(* Schneider Machine Expert - Basic project control, file version 2.7.0.0 *)
(* ProjectInformations: Name=Nuevo proyecto *)

HARDWARE
  Cpu 0: TM221M16R/G
  EthernetConfiguration: NetworkName=M221, IpAllocationMode=FixedAddress, IpAddress=0.0.0.0, SubnetMask=0.0.0.0
  SerialLineConfiguration: Baud=Baud19200, Parity=ParityEven, DataBits=DataBits8, StopBits=StopBits1, PhysicalMedium=PhysicalMediumRs485, TransmissionMode=TransmissionModeModbusRtu, SlaveId=1, Addressing=SlaveAddressing
  MastTask: UsePeriodScanMode=true, PeriodScan=10
  FastTask: Period=255
  CpuBehavior: StartingMode=StartAsPreviousState, AutoSaveRamOnEeprom=true, WatchdogPeriod=250

SYMBOLS  (address, symbol, comment, settings)
  %MW0      ER
  %MW10     PRO
  %MW20     INT
  %MW30     ER_ACUM
  %MW40     DER_ERR
  %MW50     DER
  %MW60     ERR_PREV
  %MW100    U_OUT
  %KW1      KP  [Value=4]
  %KW2      KI  [Value=3]
  %KW3      KD  [Value=1]

POU Nuevo POU
  (* SectionNumber=1 *)

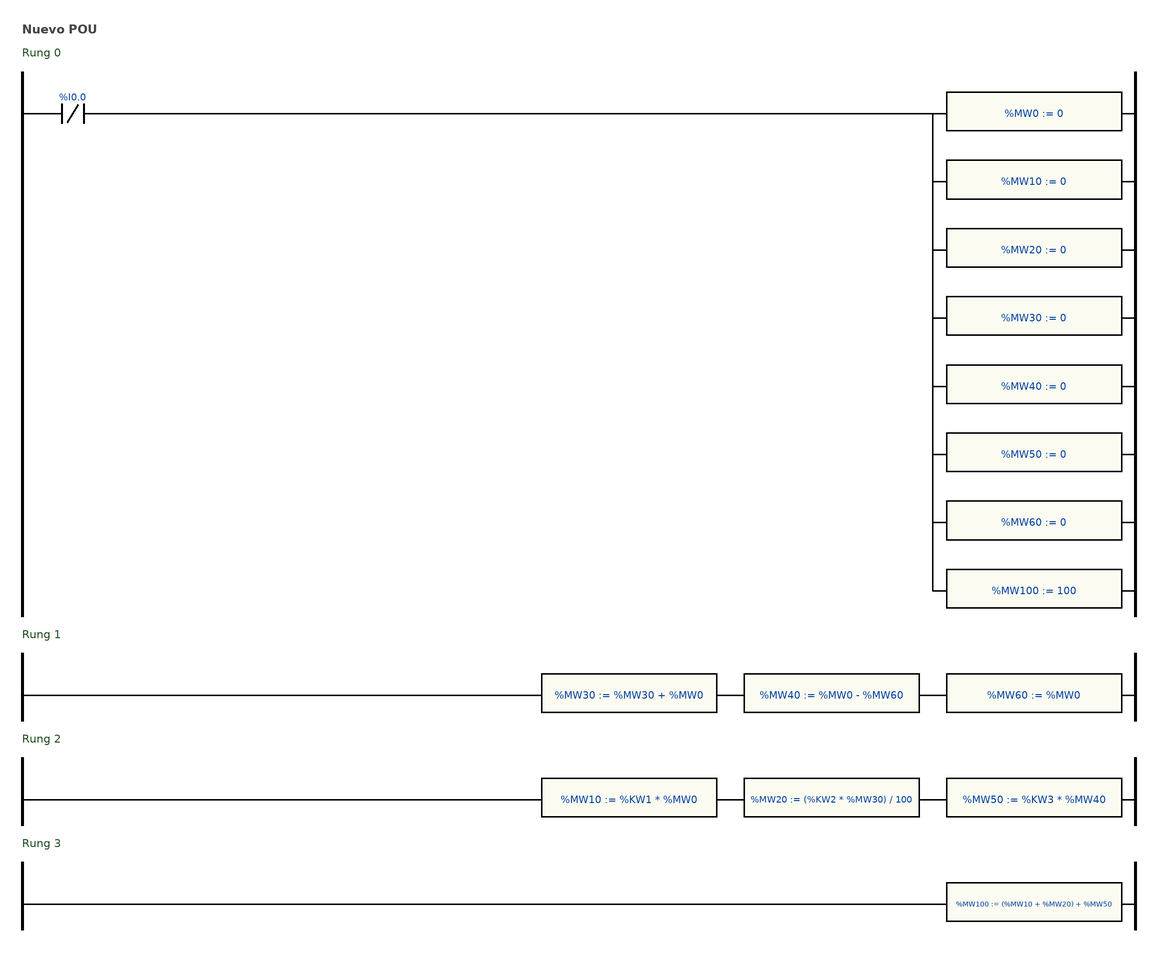

// Rung 0
  LDN %I0.0
  [ %MW0 := 0 ]           (* ER *)
  [ %MW10 := 0 ]          (* PRO *)
  [ %MW20 := 0 ]          (* INT *)
  [ %MW30 := 0 ]          (* ER_ACUM *)
  [ %MW40 := 0 ]          (* DER_ERR *)
  [ %MW50 := 0 ]          (* DER *)
  [ %MW60 := 0 ]          (* ERR_PREV *)
  [ %MW100 := 100 ]       (* U_OUT *)
  // as ST:
  //   IF NOT %I0.0 THEN ER := 0; END_IF;
  //   IF NOT %I0.0 THEN PRO := 0; END_IF;
  //   IF NOT %I0.0 THEN INT := 0; END_IF;
  //   IF NOT %I0.0 THEN ER_ACUM := 0; END_IF;
  //   IF NOT %I0.0 THEN DER_ERR := 0; END_IF;
  //   IF NOT %I0.0 THEN DER := 0; END_IF;
  //   IF NOT %I0.0 THEN ERR_PREV := 0; END_IF;
  //   IF NOT %I0.0 THEN U_OUT := 100; END_IF;

// Rung 1
  LD 1
  OPER [ %MW30 := %MW30 + %MW0 ](* ER_ACUM, ER_ACUM, ER *)
  OPER [ %MW40 := %MW0 - %MW60 ](* DER_ERR, ER, ERR_PREV *)
  [ %MW60 := %MW0 ]       (* ERR_PREV, ER *)
  // as ST:
  //   ER_ACUM := ER_ACUM + ER;
  //   DER_ERR := ER - ERR_PREV;
  //   ERR_PREV := ER;

// Rung 2
  LD 1
  OPER [ %MW10 := %KW1 * %MW0 ](* PRO, KP, ER *)
  OPER [ %MW20 := ( %KW2 * %MW30 ) / 100 ](* INT, KI, ER_ACUM *)
  [ %MW50 := %KW3 * %MW40 ](* DER, KD, DER_ERR *)
  // as ST:
  //   PRO := KP * ER;
  //   INT := ( KI * ER_ACUM ) / 100;
  //   DER := KD * DER_ERR;

// Rung 3
  LD 1
  [ %MW100 := ( %MW10 + %MW20 ) + %MW50 ](* U_OUT, PRO, INT, DER *)
  // as ST:
  //   U_OUT := ( PRO + INT ) + DER;
